// TIA Portal V20 export
TYPE "UDT_Service_Command"
   STRUCT
      reset : Bool;
      start : Bool;
      stop : Bool;
      hold : Bool;
      unhold : Bool;
      pause : Bool;
      resume : Bool;
      abort : Bool;
      restart : Bool;
      complete : Bool;
   END_STRUCT;
END_TYPE
